// TwinCAT 3 PLC project xPPU_Lib
// Title: xPPU
// Company: Jan Wilch
// ProjectVersion: 1.0.0
// ProgramVersion: 3.1.4026.11
// libraries:
//   Tc2_Standard, * (Beckhoff Automation GmbH)
//   Tc2_System, * (Beckhoff Automation GmbH)
//   Tc3_Module, * (Beckhoff Automation GmbH)
//   [Resi4MPM], * (Jan Wilch)
// project tree:
//   03_ControlPrimitives/Carrier/Crane/ Crane_MoveBase.TcPOU (not stored), Crane_MoveToLSC.TcPOU (not stored), Crane_MoveToStack.TcPOU (not stored), Crane_MoveToStamp.TcPOU (not stored), Crane_PickPutBase.TcPOU (not stored), Crane_PickUpWP.TcPOU (not stored), Crane_PutDownWP.TcPOU (not stored)
//   03_ControlPrimitives/Carrier/PickAlpha/ PicAlpha_MoveBase.TcPOU (not stored), PicAlpha_MoveToPos1.TcPOU (not stored), PicAlpha_MoveToPos2.TcPOU (not stored), PicAlpha_MoveToPos3.TcPOU (not stored), PicAlpha_MoveToPos4.TcPOU (not stored), PicAlpha_PickUpWP.TcPOU (not stored), PicAlpha_PutDownWP.TcPOU (not stored)
//   03_ControlPrimitives/Conveyor/LSC/ LSC_MoveWorkpiece_Base.TcPOU (not stored), LSC_SearchWorkpiece.TcPOU (not stored), LSC_TransferWorkpieceTo_PAC.TcPOU, LSC_TransferWorkpieceTo_RampEnd.TcPOU (not stored), LSC_TransferWorkpieceTo_RampMid.TcPOU (not stored), LSC_TransferWorkpieceTo_RampStart.TcPOU (not stored), LSC_TransferWPAtStart.TcPOU (not stored)
//   03_ControlPrimitives/Conveyor/PAC/ PAC_MoveWorkpiece_Base.TcPOU (not stored), PAC_TransferFirstWorkpieceTo_SSCStart.TcPOU (not stored), PAC_TransferWorkpieceTo_PSStart.TcPOU (not stored), PAC_TransferWorkpieceTo_SSC.TcPOU
//   03_ControlPrimitives/Conveyor/RFC/ RFC_MoveWorkpiece_Base.TcPOU (not stored), RFC_TransferWorkpieceTo_LSC.TcPOU (not stored), RFC_TransferWorkpieceTo_PSEnd.TcPOU (not stored)
//   03_ControlPrimitives/Conveyor/SSC/ SSC_MoveWorkpieceTo_PSEnd.TcPOU, SSC_MoveWorkpiece_Base.TcPOU (not stored), SSC_TransferWorkpieceTo_PSStart.TcPOU (not stored), SSC_TransferWorkpieceTo_RampEnd.TcPOU, SSC_TransferWorkpieceTo_RFC.TcPOU (not stored)
//   03_ControlPrimitives/Generic/ Delay.TcPOU (not stored), ForceProcessVariable.TcPOU (not stored), IndicateActivity.TcPOU (not stored)
//   03_ControlPrimitives/Stack/ Stack_ProvideWorkpiece.TcPOU (not stored)
//   03_ControlPrimitives/Stamp/ Stamp_StampWorkpiece.TcPOU (not stored)
//   04_HardwareObservation/ ObserveCrane.TcPOU (not stored), ObserveLSC.TcPOU (not stored), ObservePAC.TcPOU (not stored), ObservePicAlpha.TcPOU (not stored), ObserveRFC.TcPOU (not stored), ObserveSSC.TcPOU, ObserveStack.TcPOU (not stored), ObserveStamp.TcPOU (not stored), xPPUProduct.TcPOU
//   05_HardwareControl/ControlModule/ BaseComponent.TcPOU (not stored), Motor.TcPOU (not stored)
//   05_HardwareControl/ControlModule/Gen/ ActivityIndicator.TcPOU (not stored)
//   05_HardwareControl/ControlModule/Grippers/ BaseGripper.TcPOU (not stored), VacuumGripper.TcPOU (not stored)
//   05_HardwareControl/ControlModule/Pushers/ BaseCylinder.TcPOU (not stored), BistableCylinder.TcPOU (not stored), MonostableCylinder.TcPOU (not stored), Switch.TcPOU (not stored)
//   05_HardwareControl/ControlModule/Sensors/ InductiveSensor.TcPOU (not stored), OpticalSensor.TcPOU (not stored), PresenceSensor.TcPOU (not stored), PressureSensor.TcPOU (not stored), WeightSensor.TcPOU (not stored)
//   05_HardwareControl/ControlModule/Valves/ PropotionalValve.TcPOU (not stored)
//   05_HardwareControl/DUTs/ ActuatorConfiguration.TcDUT (not stored), BaseConfiguration.TcDUT (not stored), ConveyorConfiguration.TcDUT (not stored), ConveyorOutput.TcDUT (not stored), EWPMaterial.TcDUT (not stored), EWPWeight.TcDUT (not stored), MotorOutput.TcDUT (not stored), RampConfiguration.TcDUT (not stored), SensorConfiguration.TcDUT (not stored), SensorOutput.TcDUT (not stored)
//   05_HardwareControl/EquipmentModule/Carriers/ BaseCarrier.TcPOU (not stored), Crane.TcPOU (not stored), PicAlpha.TcPOU (not stored)
//   05_HardwareControl/EquipmentModule/Conveyors/ Conveyor.TcPOU (not stored), LargeSortingConveyor.TcPOU (not stored), PicAlphaConveyor.TcPOU (not stored), RefeedingConveyor.TcPOU (not stored), SmallSortingConveyor.TcPOU (not stored)
//   05_HardwareControl/EquipmentModule/Ramps/ Ramp.TcPOU (not stored)
//   05_HardwareControl/EquipmentModule/Stacks/ Stack.TcPOU (not stored)
//   05_HardwareControl/EquipmentModule/Stamps/ Stamp.TcPOU (not stored)
//   05_HardwareControl/Interfaces/ ITF_AnalogSensor.TcIO (not stored), ITF_BinarySensor.TcIO (not stored), ITF_Cylinder.TcIO (not stored)
//   98_NamingEnums/ EAlarms.TcDUT (not stored), EOperatingModes.TcDUT (not stored), EPrimitives.TcDUT (not stored), EProcessVariables.TcDUT (not stored), EProducts.TcDUT, EProductTypes.TcDUT (not stored), ESequences.TcDUT (not stored), EStampStates.TcDUT (not stored)
//   99_ExtrafunctionalImpl/ PanelManager.TcPOU (not stored), ErrorManager.TcPOU (not stored), FC_InitAlarmTexts.TcPOU (not stored), MachineModes.TcPOU (not stored)
//   GVLs/ HMI_Texts.TcGVL (not stored)

// ---- 98_NamingEnums/EProducts.TcDUT
{attribute 'qualified_only'}
{attribute 'strict'}
TYPE EProducts :
(
	none := 0,
	stack_product := 1,
	crane_product := 2,
	stamp_product := 3,
	LSC_product := 4,
	PAC_product1 := 5,
	PAC_product2 := 6,
	PAC_product3 := 7,
	PicAlpha_product := 8,
	RFC_product1 := 9,
	RFC_product2 := 10,
	SSC_product1 := 11,
	SSC_product2 := 12,
	SSC_product3 := 13
) UINT;
END_TYPE

// ---- 03_ControlPrimitives/Conveyor/LSC/LSC_TransferWorkpieceTo_PAC.TcPOU
FUNCTION_BLOCK LSC_TransferWorkpieceTo_PAC EXTENDS LSC_MoveWorkpiece_Base
VAR_INPUT
END_VAR
VAR_OUTPUT
END_VAR
VAR
	// (EProcessVariables.PAC_WPNumber < 3) AND (((EProcessVariables.PicAlpha_AtPos1 = FALSE) AND (EProcessVariables.PicAlpha_AtPos2 = FALSE)) OR (EProcessVariables.PicAlpha_CylinderRetracted = TRUE))
	m_compExpr91: ComparisonExpression(EProcessVariables.PAC_WPNumber, EComparisonType.less, EDataType.numeric, FALSE, 3, '', TRUE);
	m_compExpr93: ComparisonExpression(EProcessVariables.PicAlpha_AtPos1, EComparisonType.equals, EDataType.binary, FALSE, 0, '', TRUE);
	m_compExpr95: ComparisonExpression(EProcessVariables.PicAlpha_AtPos2, EComparisonType.equals, EDataType.binary, FALSE, 0, '', TRUE);
	m_boolExpr96: BoolExpression(m_compExpr93, EBoolOperation.and_op, m_compExpr95);
	m_compExpr98: ComparisonExpression(EProcessVariables.PicAlpha_CylinderRetracted, EComparisonType.equals, EDataType.binary, TRUE, 0, '', TRUE);
	m_boolExpr99: BoolExpression(m_boolExpr96, EBoolOperation.or_op, m_compExpr98);
	m_precondition: BoolExpression(m_compExpr91, EBoolOperation.and_op, m_boolExpr99);
	
	// EProcessVariables.PAC_WPAtStart = TRUE
	m_postcondition: ComparisonExpression(EProcessVariables.PAC_WPAtStart, EComparisonType.equals, EDataType.binary, TRUE, 0, '', TRUE);
	
	m_timer: TON;
	//m_timerPassby : TON;
    m_timerEject  : TON;
	m_passby: BOOL;
END_VAR

SUPER^();

METHOD PROTECTED  AtTarget : BOOL
VAR_INPUT
END_VAR
AtTarget := FALSE;
m_ptrLSC^.METH_Switch_Extend();

IF m_ptrLSC^.WPAtStart THEN
	m_passby := TRUE;
END_IF

IF m_passby THEN
	m_timer(IN := TRUE, PT := T#2000MS);
	IF m_timer.Q THEN
		m_timer(IN := FALSE, PT := T#0MS);
		m_passby := FALSE;
		AtTarget := TRUE;
	END_IF
END_IF
END_METHOD

METHOD PROTECTED EjectOperation : BOOL
VAR_INPUT
END_VAR
EjectOperation := FALSE;

m_ptrLSC^.METH_Switch_Extend();
m_ptrLSC^.METH_ConveyorForward();
m_timerEject(IN := TRUE, PT := T#2000MS);

IF m_timerEject.Q THEN
  m_timerEject(IN := FALSE, PT := T#0MS);
  m_ptrLSC^.METH_Switch_Retract();
  m_ptrLSC^.METH_ConveyorStop();
  EjectOperation := TRUE;
END_IF
END_METHOD

METHOD FB_init : BOOL
VAR_INPUT
	bInitRetains : BOOL; // if TRUE, the retain variables are initialized (warm start / cold start)
	bInCopyCode : BOOL;  // if TRUE, the instance afterwards gets moved into the copy code (online change)
	
	i_ptrLSC: POINTER TO LargeSortingConveyor;
END_VAR
m_ptrLSC := i_ptrLSC;

m_id := EPrimitives.LSC_TransferWorkpieceTo_PAC;
m_timeout := T#5S;

Precondition := m_precondition;
Postcondition := m_postcondition;
END_METHOD

END_FUNCTION_BLOCK

// ---- 03_ControlPrimitives/Conveyor/PAC/PAC_TransferWorkpieceTo_SSC.TcPOU
FUNCTION_BLOCK PAC_TransferWorkpieceTo_SSC EXTENDS PAC_MoveWorkpiece_Base
VAR_INPUT
	i_ptrSSC : POINTER TO SmallSortingConveyor;
END_VAR
VAR_OUTPUT
END_VAR
VAR
	 m_ptrSSC    : POINTER TO SmallSortingConveyor;
	// (EProcessVariables.PicAlpha_AtPos3 = TRUE) AND ((EProcessVariables.PicAlpha_HoldingWorkpiece = FALSE) AND ((EProcessVariables.PicAlpha_CylinderRetracted = TRUE) AND ((EProcessVariables.PAC_WPAtStart = FALSE) AND ((EProcessVariables.SSC_ProductType_1 = 0) AND (EProcessVariables.SSC_ProductType_2 = 0)))))
	m_compExpr127: ComparisonExpression(EProcessVariables.PicAlpha_AtPos3, EComparisonType.equals, EDataType.binary, TRUE, 0, '', TRUE);
	m_compExpr129: ComparisonExpression(EProcessVariables.PicAlpha_HoldingWorkpiece, EComparisonType.equals, EDataType.binary, FALSE, 0, '', TRUE);
	m_compExpr131: ComparisonExpression(EProcessVariables.PicAlpha_CylinderRetracted, EComparisonType.equals, EDataType.binary, TRUE, 0, '', TRUE);
	m_compExpr133: ComparisonExpression(EProcessVariables.PAC_WPAtStart, EComparisonType.equals, EDataType.binary, FALSE, 0, '', TRUE);
	m_compExpr135: ComparisonExpression(EProcessVariables.SSC_ProductType_1, EComparisonType.equals, EDataType.numeric, FALSE, 0, '', TRUE);
	m_compExpr137: ComparisonExpression(EProcessVariables.SSC_ProductType_2, EComparisonType.equals, EDataType.numeric, FALSE, 0, '', TRUE);
	m_boolExpr138: BoolExpression(m_compExpr135, EBoolOperation.and_op, m_compExpr137);
	m_boolExpr139: BoolExpression(m_compExpr133, EBoolOperation.and_op, m_boolExpr138);
	m_boolExpr140: BoolExpression(m_compExpr131, EBoolOperation.and_op, m_boolExpr139);
	m_boolExpr141: BoolExpression(m_compExpr129, EBoolOperation.and_op, m_boolExpr140);
	m_precondition: BoolExpression(m_compExpr127, EBoolOperation.and_op, m_boolExpr141);
	
	// EProcessVariables.PAC_WPAtEnd = FALSE
	m_postcondition: ComparisonExpression(EProcessVariables.PAC_WPAtEnd, EComparisonType.equals, EDataType.binary, FALSE, 0, '', TRUE);
	
	m_timer : TON;
END_VAR

SUPER^();

METHOD PROTECTED  AtTarget : BOOL
VAR_INPUT
END_VAR
AtTarget := FALSE;
IF NOT m_ptrPAC^.WPAtEnd THEN
	m_timer(IN := TRUE, PT := T#1500MS);
	IF m_timer.Q THEN
		m_timer(IN := FALSE);
		m_ptrPAC^.METH_ResetWPNumberAtPAC();
		AtTarget := TRUE;
	END_IF
END_IF
END_METHOD

METHOD PROTECTED EjectOperation : BOOL
VAR_INPUT
END_VAR
EjectOperation := TRUE;
END_METHOD

METHOD FB_init : BOOL
VAR_INPUT
	bInitRetains : BOOL; // if TRUE, the retain variables are initialized (warm start / cold start)
	bInCopyCode : BOOL;  // if TRUE, the instance afterwards gets moved into the copy code (online change)
	
	i_ptrPAC: POINTER TO PicAlphaConveyor;
END_VAR
m_ptrPAC := i_ptrPAC;

 SUPER^(); //
  m_ptrSSC := i_ptrSSC; //      
  FB_init := TRUE; //

m_id := EPrimitives.PAC_TransferWorkpieceTo_SSC;
m_timeout := T#200S;

Precondition := m_precondition;
Postcondition := m_postcondition;
END_METHOD

END_FUNCTION_BLOCK

// ---- 03_ControlPrimitives/Conveyor/SSC/SSC_MoveWorkpieceTo_PSEnd.TcPOU
FUNCTION_BLOCK SSC_MoveWorkpieceTo_PSEnd EXTENDS SSC_MoveWorkpiece_Base
VAR_INPUT
END_VAR
VAR_OUTPUT
END_VAR
VAR

// (EProcessVariables.PicAlpha_AtPos3 = TRUE) AND ((EProcessVariables.PicAlpha_HoldingWorkpiece = FALSE) AND (EProcessVariables.PicAlpha_CylinderExtended = FALSE))
	m_compExpr244: ComparisonExpression(EProcessVariables.PAC_WPAtEnd, EComparisonType.equals, EDataType.binary, TRUE, 0, '', TRUE);
	m_compExpr246: ComparisonExpression(EProcessVariables.PicAlpha_HoldingWorkpiece, EComparisonType.equals, EDataType.binary, FALSE, 0, '', TRUE);
	m_compExpr248: ComparisonExpression(EProcessVariables.PicAlpha_CylinderRetracted, EComparisonType.equals, EDataType.binary, TRUE, 0, '', TRUE);
	//m_compExpr250: ComparisonExpression(EProcessVariables.RFC_ProductType_1, EComparisonType.equals, EDataType.numeric, FALSE, 0, '', TRUE);
	//m_compExpr252: ComparisonExpression(EProcessVariables.RFC_ProductType_2, EComparisonType.equals, EDataType.numeric, FALSE, 0, '', TRUE);
	//m_boolExpr253: BoolExpression(m_compExpr250, EBoolOperation.and_op, m_compExpr252);
	//m_boolExpr254: BoolExpression(m_compExpr248, EBoolOperation.and_op, m_boolExpr253);
	m_boolExpr255: BoolExpression(m_compExpr246, EBoolOperation.and_op, m_compExpr248);
	m_precondition: BoolExpression(m_compExpr244, EBoolOperation.and_op, m_boolExpr255);
	m_postcondition: ValueExpression(EDataType.binary, TRUE, 0, '', TRUE);
	
	m_timer: TON;
	m_passby : BOOL;

END_VAR

SUPER^();

METHOD PROTECTED AtTarget : BOOL
VAR_INPUT
END_VAR
AtTarget := FALSE;

IF m_ptrSSC^.WPAtEnd THEN
	AtTarget := TRUE;
END_IF
END_METHOD

{warning 'Methodenimplementierung hinzufügen'}
METHOD PROTECTED EjectOperation : BOOL
EjectOperation := TRUE;
END_METHOD

//FB_Init ist immer implizit verfügbar und wird primär für die Initialisierung verwendet.
//Der Rückgabewert wird nicht ausgewertet. Für gezielte Einflussnahme können Sie
//die Methoden explizit deklarieren und darin mit dem Standard-Initialisierungscode 
//zusätzlichen Code bereitstellen. Sie können den Rückgabewert auswerten.
METHOD FB_Init: BOOL
VAR_INPUT    
bInitRetains: BOOL; // TRUE: Die Retain-Variablen werden initialisiert (Reset warm / Reset kalt)    
bInCopyCode: BOOL;  // TRUE: Die Instanz wird danach in den Kopiercode kopiert (Online-Change)
i_ptrSSC: POINTER TO SmallSortingConveyor;
END_VAR
VAR
END_VAR
//m_ptrSSC := i_ptrSSC;

m_id := EPrimitives.SSC_TransferWorkpieceTo_RFC;
m_timeout := T#200S;

Precondition := m_precondition;
Postcondition := m_postcondition;

FB_init := TRUE;
END_METHOD

END_FUNCTION_BLOCK

// ---- 03_ControlPrimitives/Conveyor/SSC/SSC_TransferWorkpieceTo_RampEnd.TcPOU
FUNCTION_BLOCK SSC_TransferWorkpieceTo_RampEnd EXTENDS SSC_MoveWorkpiece_Base
VAR_INPUT
END_VAR
VAR_OUTPUT
END_VAR
VAR
	// (EProcessVariables.PicAlpha_AtPos3 = TRUE) AND ((EProcessVariables.PicAlpha_HoldingWorkpiece = FALSE) AND (EProcessVariables.PicAlpha_CylinderExtended = FALSE))
	m_compExpr233: ComparisonExpression(EProcessVariables.PicAlpha_AtPos3, EComparisonType.equals, EDataType.binary, TRUE, 0, '', TRUE);
	m_compExpr235: ComparisonExpression(EProcessVariables.PicAlpha_HoldingWorkpiece, EComparisonType.equals, EDataType.binary, FALSE, 0, '', TRUE);
	m_compExpr237: ComparisonExpression(EProcessVariables.PicAlpha_CylinderExtended, EComparisonType.equals, EDataType.binary, FALSE, 0, '', TRUE);
	m_boolExpr238: BoolExpression(m_compExpr235, EBoolOperation.and_op, m_compExpr237);
	m_precondition: BoolExpression(m_compExpr233, EBoolOperation.and_op, m_boolExpr238);
	
	// TRUE
	m_postcondition: ValueExpression(EDataType.binary, TRUE, 0, '', TRUE);
	
	m_timer: TON;
	m_passby : BOOL;
END_VAR

SUPER^();

METHOD PROTECTED  AtTarget : BOOL
VAR_INPUT
END_VAR
AtTarget := FALSE;

IF m_ptrSSC^.WPAtRampEnd THEN
	m_passby := TRUE;
END_IF

IF m_passby THEN
	m_timer(IN := TRUE, PT := T#500MS);
	IF m_timer.Q THEN
		m_timer(IN := FALSE);
		m_passby := FALSE;
		AtTarget := TRUE;
	END_IF
END_IF
END_METHOD

METHOD PROTECTED EjectOperation : BOOL
VAR_INPUT
END_VAR
EjectOperation := TRUE;
END_METHOD

METHOD FB_init : BOOL
VAR_INPUT
	bInitRetains : BOOL; // if TRUE, the retain variables are initialized (warm start / cold start)
	bInCopyCode : BOOL;  // if TRUE, the instance afterwards gets moved into the copy code (online change)
	
	i_ptrSSC: POINTER TO SmallSortingConveyor;
END_VAR
m_ptrSSC := i_ptrSSC;
m_passby := FALSE;

m_id := EPrimitives.SSC_TransferWorkpieceTo_RampEnd;
m_timeout := T#200S;

Precondition := m_precondition;
Postcondition := m_postcondition;

FB_init := TRUE;
END_METHOD

END_FUNCTION_BLOCK

// ---- 04_HardwareObservation/ObserveSSC.TcPOU
FUNCTION_BLOCK ObserveSSC EXTENDS HardwareObservationBase
VAR_INPUT
END_VAR
VAR_OUTPUT
END_VAR
VAR
	m_ptrSSC: POINTER TO SmallSortingConveyor;
	m_ptrSSCWP1: POINTER TO xPPUProduct;
	m_ptrSSCWP2: POINTER TO xPPUProduct;
	m_ptrSSCWP3: POINTER TO xPPUProduct;
	m_rtWpAtRamp: R_TRIG;
END_VAR

METHOD FB_init : BOOL
VAR_INPUT
	bInitRetains : BOOL; // if TRUE, the retain variables are initialized (warm start / cold start)
	bInCopyCode : BOOL;  // if TRUE, the instance afterwards gets moved into the copy code (online change)
	
	i_ptrSSC: POINTER TO SmallSortingConveyor;
	i_ptrWP1: POINTER TO xPPUProduct;
	i_ptrWP2: POINTER TO xPPUProduct;
	i_ptrWP3: POINTER TO xPPUProduct;
END_VAR
m_ptrSSC := i_ptrSSC;
m_ptrSSCWP1 := i_ptrWP1;
m_ptrSSCWP2 := i_ptrWP2;
m_ptrSSCWP3 := i_ptrWP3;
END_METHOD

METHOD  ResetDefinition : BOOL
VAR_INPUT
END_VAR
;
END_METHOD

(* Update an instance of ProcessState with the part of the process that can be observed by this Hardware Interface. *)
METHOD UpdateProcessObservation : BOOL
VAR_IN_OUT
	io_processState: ProcessState;
END_VAR
m_rtWpAtRamp(CLK := m_ptrSSC^.WPAtRampEnd);

io_processState.UpdateState_Binary(EProcessVariables.SSC_WPAtStart, m_ptrSSC^.WPAtStart, TRUE);
io_processState.UpdateState_Binary(EProcessVariables.SSC_WPAtEnd, m_ptrSSC^.WPAtEnd, TRUE);
io_processState.UpdateState_Binary(EProcessVariables.SSC_WPLightAtMiddle, m_ptrSSC^.LightWPAtMid, TRUE);
io_processState.UpdateState_Binary(EProcessVariables.SSC_WPMetalAtMiddle, m_ptrSSC^.MetalWPAtMid, TRUE);
io_processState.UpdateState_Binary(EProcessVariables.SSC_WPAtRampEnd, m_ptrSSC^.WPAtRampEnd, TRUE);
io_processState.UpdateState_Binary(EProcessVariables.SSC_SwitchExtended, m_ptrSSC^.m_Switch.Extended, TRUE);
io_processState.UpdateState_Binary(EProcessVariables.SSC_SwitchRetracted, m_ptrSSC^.m_Switch.Retracted, TRUE);

IF m_rtWpAtRamp.Q THEN
	io_processState.UpdateState_NumericIncrement(EProcessVariables.SSC_RampWPCount, TRUE);
END_IF


io_processState.UpdateState_Defined(EProcessVariables.SSC_WPAtStart, TRUE);
io_processState.UpdateState_Defined(EProcessVariables.SSC_WPAtEnd, TRUE);
io_processState.UpdateState_Defined(EProcessVariables.SSC_WPLightAtMiddle, TRUE);
io_processState.UpdateState_Defined(EProcessVariables.SSC_WPMetalAtMiddle, TRUE);
io_processState.UpdateState_Defined(EProcessVariables.SSC_WPAtRampEnd, TRUE);
io_processState.UpdateState_Defined(EProcessVariables.SSC_SwitchExtended, TRUE);
io_processState.UpdateState_Defined(EProcessVariables.SSC_SwitchRetracted, TRUE);
// TODO - the following is technically not defined but how can we avoid that?
io_processState.UpdateState_Defined(EProcessVariables.SSC_RampWPCount, TRUE);
END_METHOD

END_FUNCTION_BLOCK

// ---- 04_HardwareObservation/xPPUProduct.TcPOU
FUNCTION_BLOCK xPPUProduct EXTENDS ProductBase
VAR CONSTANT
	LIGHT_IDX: USINT := 1;
	METAL_IDX: USINT := 2;
	PRESENT_IDX: USINT := 3;
END_VAR

//FB_Init is always available implicitly and it is used primarily for initialization.
//The return value is not evaluated. For a specific influence, you can also declare the
//methods explicitly and provide additional code there with the standard initialization
//code. You can evaluate the return value.
METHOD FB_Init: BOOL
VAR_INPUT
    bInitRetains: BOOL; // TRUE: the retain variables are initialized (reset warm / reset cold)
    bInCopyCode: BOOL;  // TRUE: the instance will be copied to the copy code afterward (online change)
	
	i_productTypeVarId: UINT;
END_VAR
// set the variable indices (on remote, the RA does this)
raIn_processStateIdx := i_productTypeVarId;

// set the variables' data types
m_vals[RES_IDX].DataType := EDataType.numeric;
m_vals[LIGHT_IDX].DataType := EDataType.binary;
m_vals[METAL_IDX].DataType := EDataType.binary;
m_vals[PRESENT_IDX].DataType := EDataType.binary;
END_METHOD

PROPERTY IsLight : BOOL
GET
IsLight := m_vals[LIGHT_IDX].Defined AND m_vals[LIGHT_IDX].Value.Binary;
END_GET
SET
m_vals[LIGHT_IDX].DataType := EDataType.binary;
m_vals[LIGHT_IDX].Defined := TRUE;
m_vals[LIGHT_IDX].Value.Binary := IsLight;

UpdateMaterial();
END_SET
END_PROPERTY

PROPERTY IsMetal : BOOL
GET
IsMetal := m_vals[METAL_IDX].Defined AND m_vals[METAL_IDX].Value.Binary;
END_GET
SET
m_vals[METAL_IDX].DataType := EDataType.binary;
m_vals[METAL_IDX].Defined := TRUE;
m_vals[METAL_IDX].Value.Binary := IsMetal;

UpdateMaterial();
END_SET
END_PROPERTY

PROPERTY IsPresent : BOOL
GET
IsPresent := m_vals[PRESENT_IDX].Defined AND m_vals[PRESENT_IDX].Value.Binary;
END_GET
SET
m_vals[PRESENT_IDX].DataType := EDataType.binary;
m_vals[PRESENT_IDX].Defined := TRUE;
m_vals[PRESENT_IDX].Value.Binary := IsPresent;

UpdateMaterial();
END_SET
END_PROPERTY

(* Based on the aggregated product type value, set the separete input values for a consistent shift register. *)
METHOD ReverseSetInputs : BOOL
VAR
	prodType: EProductTypes;
END_VAR
prodType := LREAL_TO_UINT(m_vals[RES_IDX].Value.Numeric);

m_vals[LIGHT_IDX].Defined := TRUE;
m_vals[METAL_IDX].Defined := TRUE;
m_vals[PRESENT_IDX].Defined := TRUE;

CASE prodType OF
	EProductTypes.none:
		m_vals[LIGHT_IDX].Value.Binary := FALSE;
		m_vals[METAL_IDX].Value.Binary := FALSE;
		m_vals[PRESENT_IDX].Value.Binary := FALSE;

// TODO - this needs a better solution...
// 	EProductTypes.unknown:
// 		m_vals[m_isLightIdx].Value.Binary := FALSE;
// 		m_vals[m_isMetalIdx].Value.Binary := FALSE;
// 		m_vals[m_isPresentIdx].Value.Binary := TRUE;
	
	EProductTypes.white:
		m_vals[LIGHT_IDX].Value.Binary := TRUE;
		m_vals[METAL_IDX].Value.Binary := FALSE;
		m_vals[PRESENT_IDX].Value.Binary := TRUE;
	EProductTypes.black:
		m_vals[LIGHT_IDX].Value.Binary := FALSE;
		m_vals[METAL_IDX].Value.Binary := FALSE;
		m_vals[PRESENT_IDX].Value.Binary := TRUE;
	EProductTypes.metal:
		m_vals[LIGHT_IDX].Value.Binary := TRUE;
		m_vals[METAL_IDX].Value.Binary := TRUE;
		m_vals[PRESENT_IDX].Value.Binary := TRUE;
	EProductTypes.unknown:
		m_vals[LIGHT_IDX].Value.Binary := FALSE;
		m_vals[METAL_IDX].Value.Binary := TRUE;
		m_vals[PRESENT_IDX].Value.Binary := TRUE;
END_CASE
END_METHOD

METHOD PRIVATE UpdateMaterial : BOOL
VAR_INPUT
END_VAR
m_vals[RES_IDX].DataType := EDataType.numeric;
m_vals[RES_IDX].Defined := TRUE;

IF IsPresent AND IsLight AND NOT IsMetal THEN
	m_vals[RES_IDX].Value.Numeric := EProductTypes.white;
ELSIF IsPresent AND NOT IsLight AND NOT IsMetal THEN
	m_vals[RES_IDX].Value.Numeric := EProductTypes.black;
ELSIF IsPresent AND IsLight AND IsMetal THEN
	m_vals[RES_IDX].Value.Numeric := EProductTypes.metal;
ELSIF IsPresent THEN
	m_vals[RES_IDX].Value.Numeric := EProductTypes.unknown;
ELSE
	m_vals[RES_IDX].Value.Numeric := EProductTypes.none;
END_IF
END_METHOD

END_FUNCTION_BLOCK
